(* Logix 5000 project; controller Test_PID 1769-L16ER-BB1B rev 32.13; software revision 32.02 *)

TASK MainTask (continuous, watchdog 500 ms) : MainProgram

MODULES
   Local : 1769-L16ER-BB1B (PointIO 0, rev 32.13)
      Analog_Input1 : 1734-IE4C (PointIO 3, rev 3.1, Input RPI 80 ms)
      Discrete_IO : Embedded (PointIO 1, rev 32.11, Output RPI 20 ms)
      Relay_Output1 : vendor 1 type 7 code 231 (PointIO 2, rev 3.1, Output RPI 20 ms)
END_MODULES

TYPE EM_ProtoRockySequence_Int :
STRUCT
   Tmr : TIMER[64];
   StepTmr : TIMER;   // Step Timer
   PrevStepNmbr : DINT;   // Previous Step Number
   Bool : BOOL[64];
   Step : BOOL[64];
   SeqCmplt : BOOL;
   SeqActv : BOOL;
   Adsorption_Mixing : BOOL;
   Adsorption_H2OAdsorption : BOOL;
   Purge : BOOL;
   Desorption_ReverseRegen : BOOL;
   Desorption_Deep_Regen : BOOL;
   Desorption_CO2HeatingTop : BOOL;
   Desorption_CO2HeatingBottom : BOOL;
   Desorption_CO2Vacuum : BOOL;
   Regeneration_N2Heatup : BOOL;
   Regeneration_N2Regeneration : BOOL;
   measure_Moisture : BOOL;
   Regeneration_Cooling : BOOL;
   CO2_Recirculation : BOOL;
   Steam : BOOL;
END_STRUCT
END_TYPE

TYPE EM_Sequence :
STRUCT
   StepNmbr : DINT;
   SecS : DINT;
   GallonS : REAL;   // Step Gallons
   GalTog : BOOL;   // Step Show Gallons Toggle
   FaultS : BOOL;   // Sequenc Fault Status
   RunS : BOOL;   // Sequence Active Status
END_STRUCT
END_TYPE

TYPE SeqSteps :
STRUCT
   Step1 : BOOL;
   Step2 : BOOL;
   Step3 : BOOL;
   Step4 : BOOL;
END_STRUCT
END_TYPE

TYPE SeqTimers :
STRUCT
   Timer1 : TIMER;
   Timer2 : TIMER;
   Timer3 : TIMER;
END_STRUCT
END_TYPE

TYPE SeqTransition :
STRUCT
   Condition1 : BOOL;
   Condition2 : BOOL;
   Condition3 : BOOL;
END_STRUCT
END_TYPE

ADD_ON_INSTRUCTION StateControl   (* revision 1.0 *)
VAR_INPUT
   AbortC : BOOL;   // Abort Command
   Alarm : BOOL;   // Alarm Status
   Complete : BOOL;   // Complete Status
   HoldC : BOOL;   // Hold Command
   OkToAbort : BOOL;   // OK to Abort
   OkToHold : BOOL;   // OK to Hold
   OkToRestart : BOOL;   // OK to Restart
   OkToStart : BOOL;   // OK to Start
   RestartC : BOOL;   // Restart Command
   StartC : BOOL;   // Start Command
END_VAR
VAR_OUTPUT
   ABORTING : BOOL; {access Read Only}   // Aborting
   AbortP : BOOL; {access Read Only}   // Abort Permissive
   HELD : BOOL; {access Read Only}   // Held
   HoldP : BOOL; {access Read Only}   // Hold Permissive
   IDLE : BOOL; {access Read Only}   // Idle
   RESTARTING : BOOL; {access Read Only}   // Restarting
   RestartP : BOOL; {access Read Only}   // Restart Permissive
   RUNNING : BOOL; {access Read Only}   // Running
   StartP : BOOL; {access Read Only}   // Start Permissive
END_VAR
VAR_INPUT
   WaitC : BOOL;   // Wait Command
END_VAR
VAR_OUTPUT
   WAITING : BOOL; {access Read Only}   // Waiting
   STARTED : BOOL; {access Read Only}   // Started
END_VAR
VAR
   AbortS : BOOL;   // Abort Status Oneshot
   RestartS : BOOL;   // Restart Status Oneshot
   HoldS : BOOL;   // Hold Status Oneshot
   StartS : BOOL;   // Start Status Oneshot
END_VAR

ROUTINE Logic   (* ladder *)
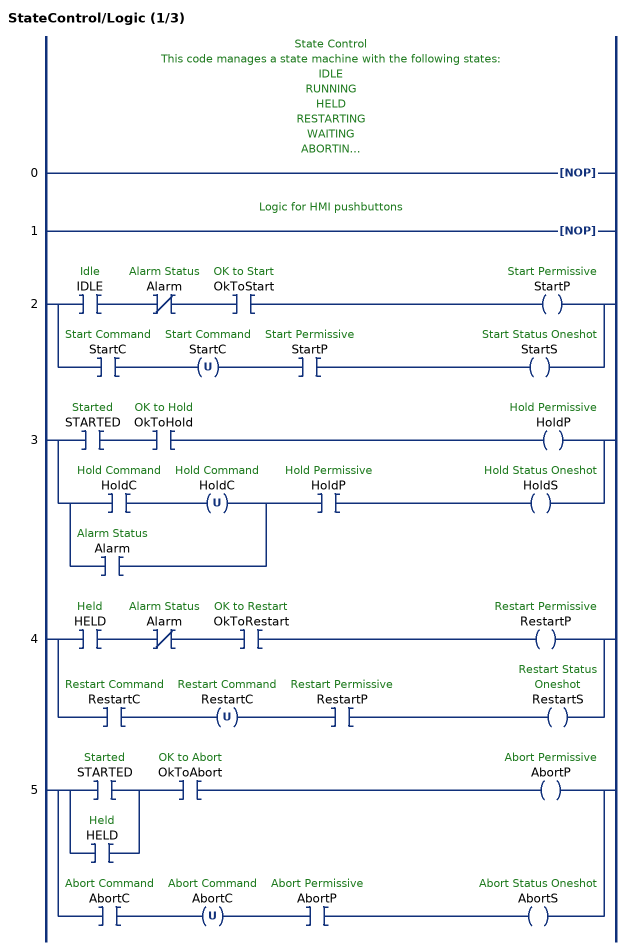
   // State Control
   // This code manages a state machine with the following states:
   // IDLE
   // RUNNING
   // HELD
   // RESTARTING
   // WAITING
   // ABORTING
   // The HMI interface consists of four pushbuttons:
   // Start
   // Hold
   // Restart
   // Abort
   // V1b - 7/15/11
   0: NOP();
   // Logic for HMI pushbuttons
   1: NOP();
   2: [XIC(IDLE) XIO(Alarm) XIC(OkToStart) OTE(StartP) ,XIC(StartC) OTU(StartC) XIC(StartP) OTE(StartS) ];
   3: [XIC(STARTED) XIC(OkToHold) OTE(HoldP) ,[XIC(HoldC) OTU(HoldC) ,XIC(Alarm) ] XIC(HoldP) OTE(HoldS) ];
   4: [XIC(HELD) XIO(Alarm) XIC(OkToRestart) OTE(RestartP) ,XIC(RestartC) OTU(RestartC) XIC(RestartP) OTE(RestartS) ];
   5: [[XIC(STARTED) ,XIC(HELD) ] XIC(OkToAbort) OTE(AbortP) ,XIC(AbortC) OTU(AbortC) XIC(AbortP) OTE(AbortS) ];
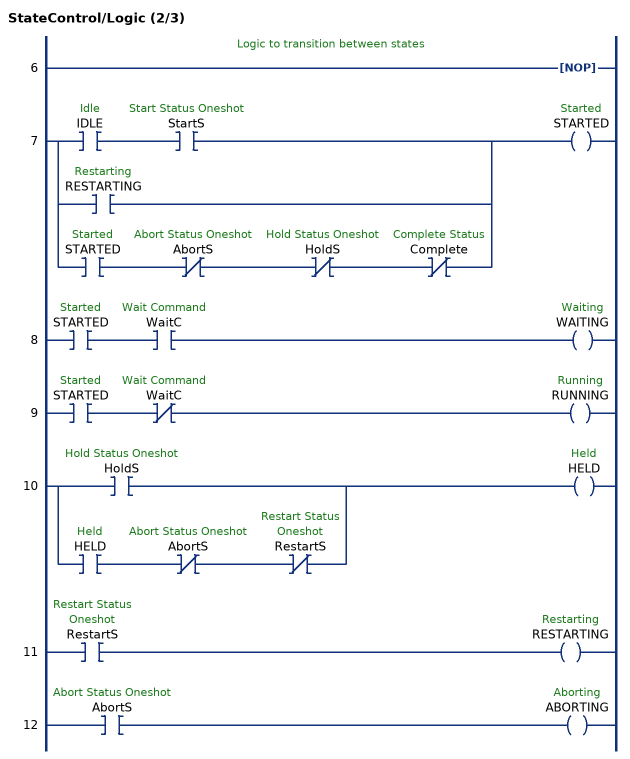
   // Logic to transition between states
   6: NOP();
   7: [[XIC(IDLE) XIC(StartS) ,XIC(RESTARTING) ] ,XIC(STARTED) XIO(AbortS) XIO(HoldS) XIO(Complete) ]OTE(STARTED);
   8: XIC(STARTED)XIC(WaitC)OTE(WAITING);
   9: XIC(STARTED)XIO(WaitC)OTE(RUNNING);
   10: [XIC(HoldS) ,XIC(HELD) XIO(AbortS) XIO(RestartS) ]OTE(HELD);
   11: XIC(RestartS)OTE(RESTARTING);
   12: XIC(AbortS)OTE(ABORTING);
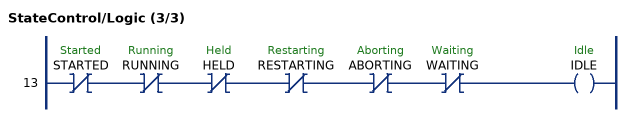
   13: XIO(STARTED)XIO(RUNNING)XIO(HELD)XIO(RESTARTING)XIO(ABORTING)XIO(WAITING)OTE(IDLE);
END_ROUTINE
END_ADD_ON_INSTRUCTION

VAR_GLOBAL   (* controller tags *)
   Alarm_Pumps_Flooding : BOOL;
   Alarm_Seq_Timeouts : BOOL;
   begin_Seq1_Start_PullDown_Tube : BOOL;
   begin_Seq3_Start_PullDown_Airlock : BOOL;
   begin_Seq4_Start_PumpDown_FS : BOOL;
   cmd_AbortPMS_HMI : BOOL;
   cmd_Close_AL_IsoV_Seq5 : BOOL;
   cmd_Close_Tube_IsoV_Seq5 : BOOL;
   cmd_FloodPumps_Seq5 : BOOL;
   cmd_Start_VentForeline : BOOL;
   cycle_type : BOOL;
   cycles_completed : DINT;
   cylcles_to_run : DINT := 3;
   emProtoRockyIISequence_i : EM_ProtoRockySequence_Int;
   emRockyIISequence : EM_Sequence;
   end_PumpsFlood_Seq : BOOL;
   fault_process : BOOL;
   Fault_Reset : BOOL;
   Fault_Seq_VentFL_Timeout : BOOL;
   hmi_abort_cycle : BOOL;
   hmi_auto_mode : BOOL := 1;
   hmi_cyles_to_run : DINT := 3;
   hmi_start_cycle : BOOL;
   hmi_stop_cycle : BOOL;
   interlockRun_VentForeline_Seq : BOOL := 1;
   interlockStart_VentForeline_Seq : BOOL := 1;
   man_seq1 : BOOL;
   man_seq11 : BOOL;
   man_seq12 : BOOL;
   man_seq13 : BOOL;
   man_seq2 : BOOL;
   man_seq3 : BOOL;
   mode_auto : BOOL := 1;
   ons_cycle_abort : BOOL;
   ons_cycle_completed : BOOL;
   ons_cycle_start : BOOL;
   ons_cycle_started : BOOL;
   ons_cycle_stop : BOOL;
   ons_seq3_done : BOOL;
   ONS_Seq_VentFL : BOOL[32];
   OpMode_isAuto : BOOL := 1;
   press_OLV_atVacuum : BOOL := 1;
   Pumps_areOFF : BOOL := 1;
   RockyIIState : StateControl := (OkToAbort := 1, OkToStart := 1, IDLE := 1, StartP := 1);
   seq11_done : BOOL;
   seq12_done : BOOL;
   seq13_done : BOOL;
   seq1_active : BOOL;
   seq1_done : BOOL;
   seq1_fault : INT;
   seq1_step : SeqSteps;
   seq1_tmr : SeqTimers := (Timer1.PRE := 10000, Timer2.PRE := 20000);
   seq1_trans : SeqTransition;
   seq2_active : BOOL;
   seq2_done : BOOL;
   seq2_fault : INT;
   seq2_step : SeqSteps;
   seq2_tmr : SeqTimers := (Timer1.PRE := 10000, Timer2.PRE := 20000);
   seq2_trans : SeqTransition;
   seq3_active : BOOL;
   seq3_done : BOOL;
   Seq_VentFL_Step : DINT;
   Seq_VentFL_StepNext : DINT;
   status_Airlock_IsoValve_isClosed : BOOL;
   status_IsoValve_isClosed : BOOL;
   status_Seq_FL_Vent_isRunning : BOOL;
   System_Faulted : BOOL;
   System_Safety_OK : BOOL := 1;
   tmr_seq_VentFL_Timeout : TIMER := (PRE := 10000);
   warning_process : BOOL;
END_VAR

PROGRAM MainProgram   (* main routine MainRoutine *)
VAR
   CO2_System_Delta_Des : DINT := 30;
   CO2Adsorption_CO2endThreshold : DINT := 10;
   PID_Loop_Call : BOOL;
   Test_Button : BOOL;
   Test_OnOff : BOOL;
   Timer_PID : TIMER := (PRE := 1000, ACC := 189, EN := 1, TT := 1);   // PID Timer
   tmr_OnOff : TIMER := (PRE := 60000);
   tmr_OnOff_Preset : DINT := 1;
END_VAR

ROUTINE Cycles_Test   (* ladder *)
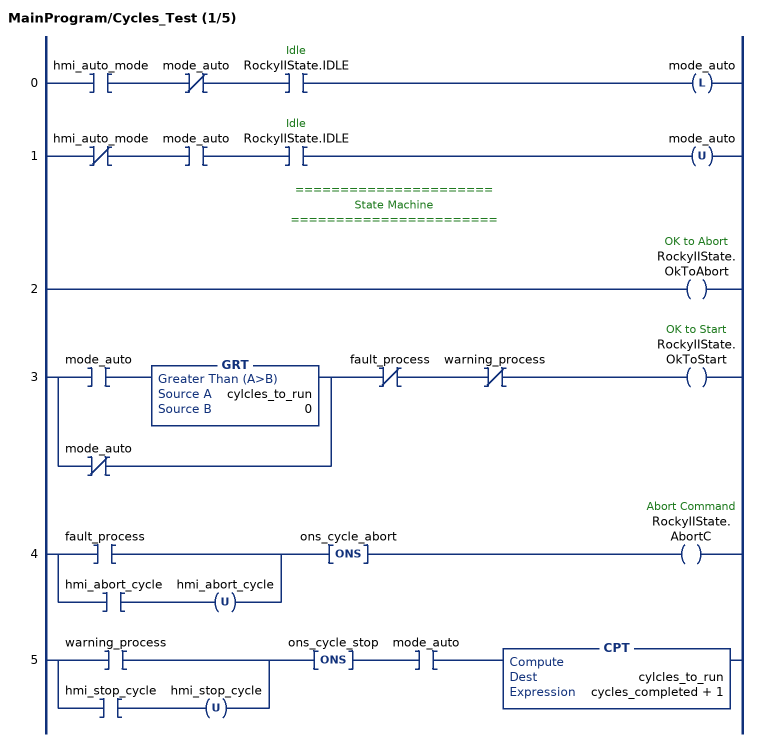
   0: XIC(hmi_auto_mode)XIO(mode_auto)XIC(RockyIIState.IDLE)OTL(mode_auto);
   1: XIO(hmi_auto_mode)XIC(mode_auto)XIC(RockyIIState.IDLE)OTU(mode_auto);
   // ======================
   // State Machine
   // =======================
   2: OTE(RockyIIState.OkToAbort);
   3: [XIC(mode_auto) GRT(cylcles_to_run,0) ,XIO(mode_auto) ]XIO(fault_process)XIO(warning_process)OTE(RockyIIState.OkToStart);
   4: [XIC(fault_process) ,XIC(hmi_abort_cycle) OTU(hmi_abort_cycle) ]ONS(ons_cycle_abort)OTE(RockyIIState.AbortC);
   5: [XIC(warning_process) ,XIC(hmi_stop_cycle) OTU(hmi_stop_cycle) ]ONS(ons_cycle_stop)XIC(mode_auto)CPT(cylcles_to_run,cycles_completed + 1);
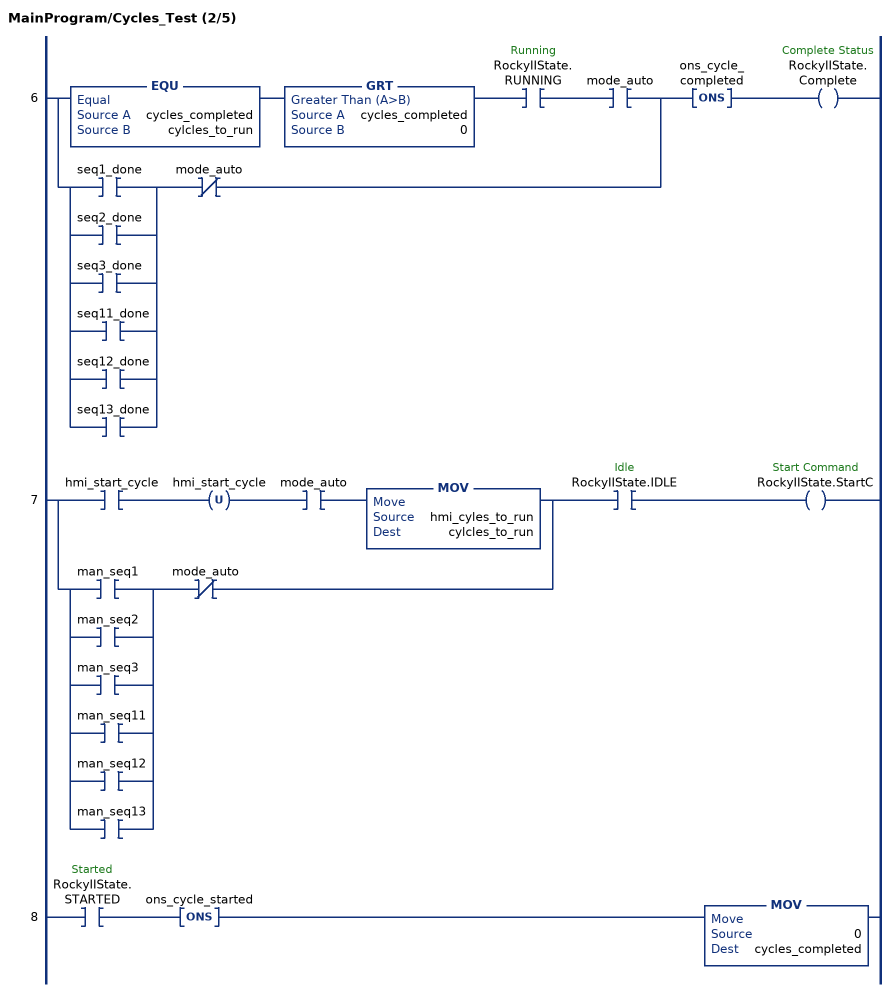
   6: [EQU(cycles_completed,cylcles_to_run) GRT(cycles_completed,0) XIC(RockyIIState.RUNNING) XIC(mode_auto) ,[XIC(seq1_done) ,XIC(seq2_done) ,XIC(seq3_done) ,XIC(seq11_done) ,XIC(seq12_done) ,XIC(seq13_done) ] XIO(mode_auto) ]ONS(ons_cycle_completed)OTE(RockyIIState.Complete);
   7: [XIC(hmi_start_cycle) OTU(hmi_start_cycle) XIC(mode_auto) MOV(hmi_cyles_to_run,cylcles_to_run) ,[XIC(man_seq1) ,XIC(man_seq2) ,XIC(man_seq3) ,XIC(man_seq11) ,XIC(man_seq12) ,XIC(man_seq13) ] XIO(mode_auto) ]XIC(RockyIIState.IDLE)OTE(RockyIIState.StartC);
   8: XIC(RockyIIState.STARTED)ONS(ons_cycle_started)MOV(0,cycles_completed);
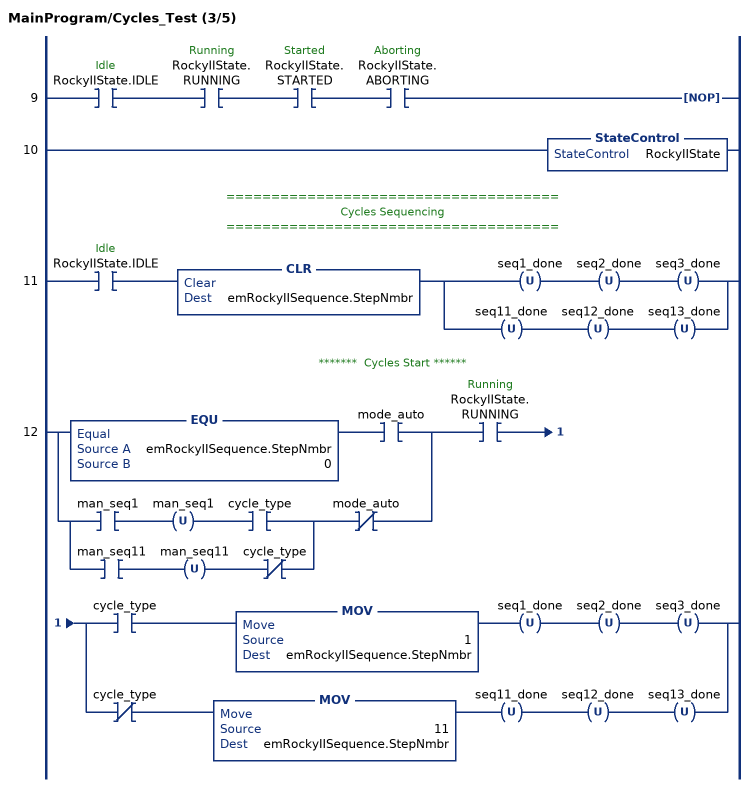
   9: XIC(RockyIIState.IDLE)XIC(RockyIIState.RUNNING)XIC(RockyIIState.STARTED)XIC(RockyIIState.ABORTING)NOP();
   10: StateControl(RockyIIState);
   // =====================================
   // Cycles Sequencing
   // =====================================
   11: XIC(RockyIIState.IDLE)CLR(emRockyIISequence.StepNmbr)[OTU(seq1_done) OTU(seq2_done) OTU(seq3_done) ,OTU(seq11_done) OTU(seq12_done) OTU(seq13_done) ];
   // *******  Cycles Start ******
   12: [EQU(emRockyIISequence.StepNmbr,0) XIC(mode_auto) ,[XIC(man_seq1) OTU(man_seq1) XIC(cycle_type) ,XIC(man_seq11) OTU(man_seq11) XIO(cycle_type) ] XIO(mode_auto) ]XIC(RockyIIState.RUNNING)[XIC(cycle_type) MOV(1,emRockyIISequence.StepNmbr) OTU(seq1_done) OTU(seq2_done) OTU(seq3_done) ,XIO(cycle_type) MOV(11,emRockyIISequence.StepNmbr) OTU(seq11_done) OTU(seq12_done) OTU(seq13_done) ];
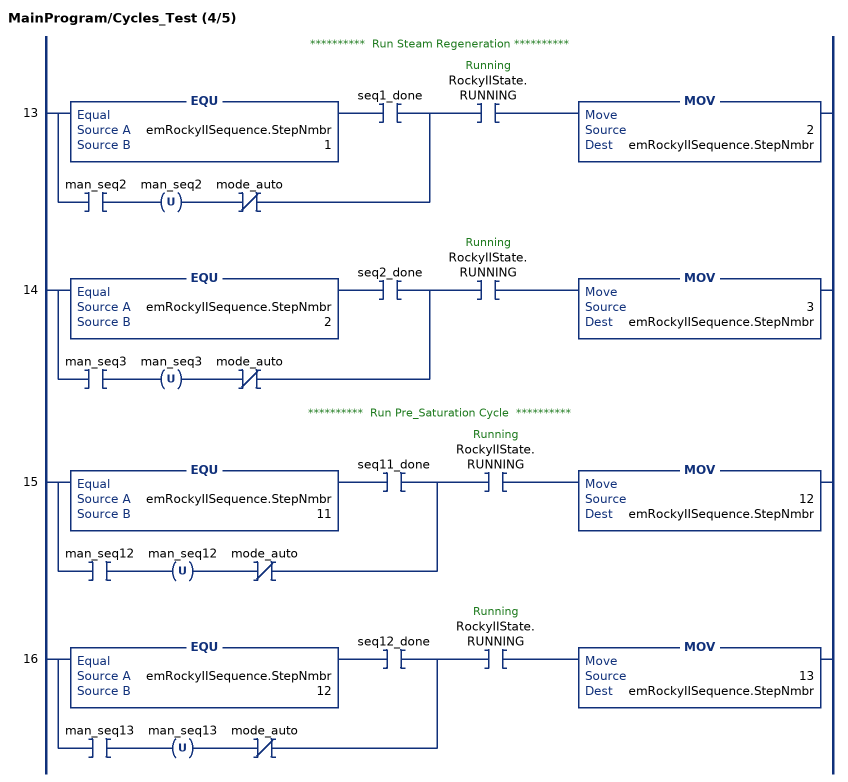
   // **********  Run Steam Regeneration **********
   13: [EQU(emRockyIISequence.StepNmbr,1) XIC(seq1_done) ,XIC(man_seq2) OTU(man_seq2) XIO(mode_auto) ]XIC(RockyIIState.RUNNING)MOV(2,emRockyIISequence.StepNmbr);
   14: [EQU(emRockyIISequence.StepNmbr,2) XIC(seq2_done) ,XIC(man_seq3) OTU(man_seq3) XIO(mode_auto) ]XIC(RockyIIState.RUNNING)MOV(3,emRockyIISequence.StepNmbr);
   // **********  Run Pre_Saturation Cycle  **********
   15: [EQU(emRockyIISequence.StepNmbr,11) XIC(seq11_done) ,XIC(man_seq12) OTU(man_seq12) XIO(mode_auto) ]XIC(RockyIIState.RUNNING)MOV(12,emRockyIISequence.StepNmbr);
   16: [EQU(emRockyIISequence.StepNmbr,12) XIC(seq12_done) ,XIC(man_seq13) OTU(man_seq13) XIO(mode_auto) ]XIC(RockyIIState.RUNNING)MOV(13,emRockyIISequence.StepNmbr);
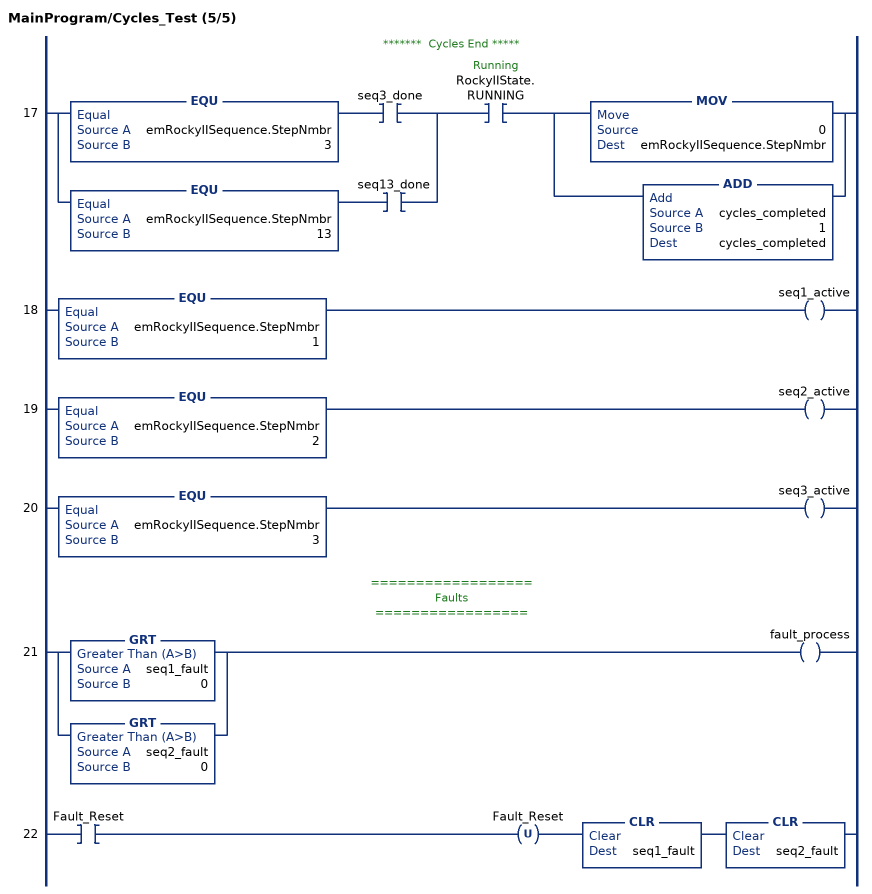
   // *******  Cycles End *****
   17: [EQU(emRockyIISequence.StepNmbr,3) XIC(seq3_done) ,EQU(emRockyIISequence.StepNmbr,13) XIC(seq13_done) ]XIC(RockyIIState.RUNNING)[MOV(0,emRockyIISequence.StepNmbr) ,ADD(cycles_completed,1,cycles_completed) ];
   18: EQU(emRockyIISequence.StepNmbr,1)OTE(seq1_active);
   19: EQU(emRockyIISequence.StepNmbr,2)OTE(seq2_active);
   20: EQU(emRockyIISequence.StepNmbr,3)OTE(seq3_active);
   // ==================
   // Faults
   // =================
   21: [GRT(seq1_fault,0) ,GRT(seq2_fault,0) ]OTE(fault_process);
   22: XIC(Fault_Reset)OTU(Fault_Reset)CLR(seq1_fault)CLR(seq2_fault);
END_ROUTINE

ROUTINE MainRoutine   (* ladder *)
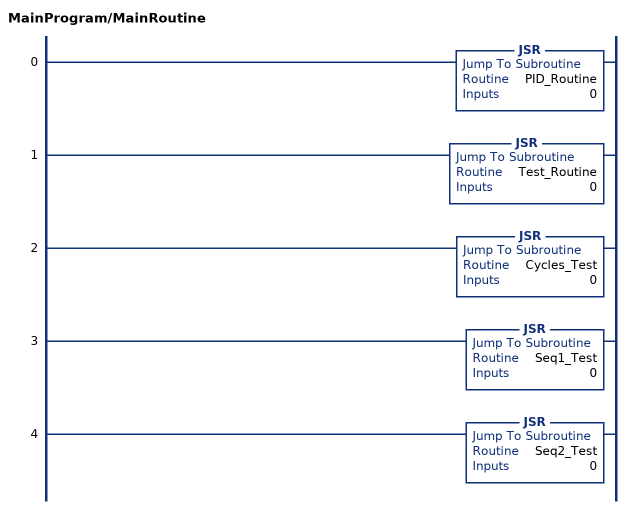
   0: JSR(PID_Routine,0);
   1: JSR(Test_Routine,0);
   2: JSR(Cycles_Test,0);
   3: JSR(Seq1_Test,0);
   4: JSR(Seq2_Test,0);
END_ROUTINE

ROUTINE PID_Routine   (* ladder *)
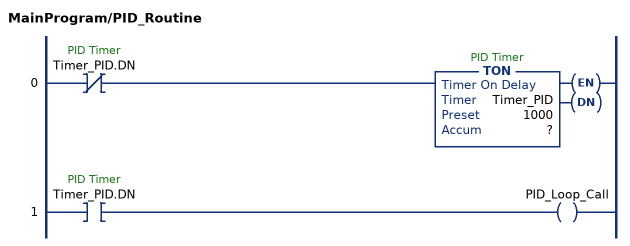
   0: XIO(Timer_PID.DN)TON(Timer_PID,?,?);
   1: XIC(Timer_PID.DN)OTE(PID_Loop_Call);
END_ROUTINE

ROUTINE Seq1_Test   (* ladder *)
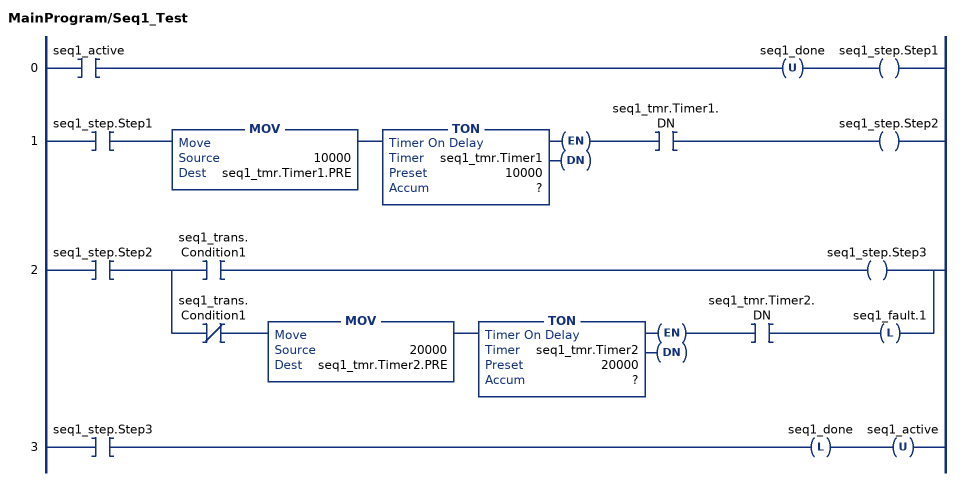
   0: XIC(seq1_active)OTU(seq1_done)OTE(seq1_step.Step1);
   1: XIC(seq1_step.Step1)MOV(10000,seq1_tmr.Timer1.PRE)TON(seq1_tmr.Timer1,?,?)XIC(seq1_tmr.Timer1.DN)OTE(seq1_step.Step2);
   2: XIC(seq1_step.Step2)[XIC(seq1_trans.Condition1) OTE(seq1_step.Step3) ,XIO(seq1_trans.Condition1) MOV(20000,seq1_tmr.Timer2.PRE) TON(seq1_tmr.Timer2,?,?) XIC(seq1_tmr.Timer2.DN) OTL(seq1_fault.1) ];
   3: XIC(seq1_step.Step3)OTL(seq1_done)OTU(seq1_active);
END_ROUTINE

ROUTINE Seq2_Test   (* ladder *)
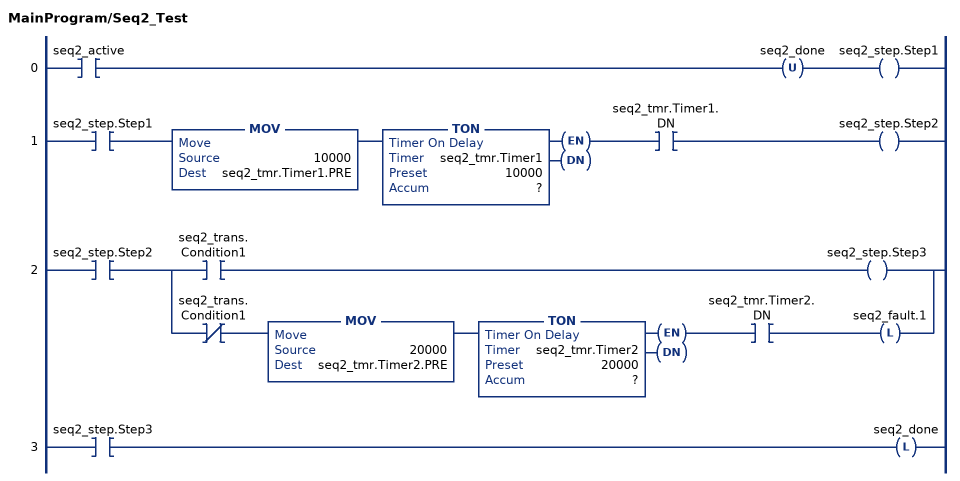
   0: XIC(seq2_active)OTU(seq2_done)OTE(seq2_step.Step1);
   1: XIC(seq2_step.Step1)MOV(10000,seq2_tmr.Timer1.PRE)TON(seq2_tmr.Timer1,?,?)XIC(seq2_tmr.Timer1.DN)OTE(seq2_step.Step2);
   2: XIC(seq2_step.Step2)[XIC(seq2_trans.Condition1) OTE(seq2_step.Step3) ,XIO(seq2_trans.Condition1) MOV(20000,seq2_tmr.Timer2.PRE) TON(seq2_tmr.Timer2,?,?) XIC(seq2_tmr.Timer2.DN) OTL(seq2_fault.1) ];
   3: XIC(seq2_step.Step3)OTL(seq2_done);
END_ROUTINE

ROUTINE Test_Routine   (* ladder *)
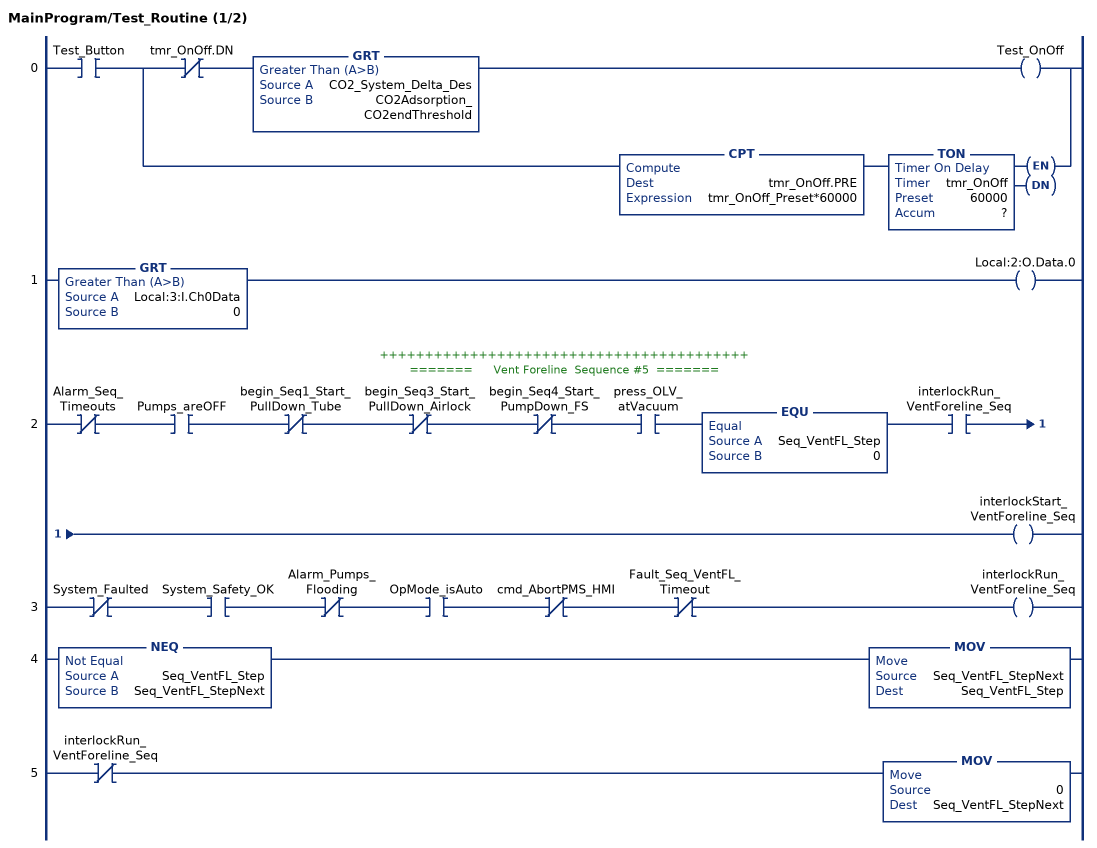
   0: XIC(Test_Button)[XIO(tmr_OnOff.DN) GRT(CO2_System_Delta_Des,CO2Adsorption_CO2endThreshold) OTE(Test_OnOff) ,CPT(tmr_OnOff.PRE,tmr_OnOff_Preset*60000) TON(tmr_OnOff,?,?) ];
   1: GRT(Local:3:I.Ch0Data,0)OTE(Local:2:O.Data.0);
   // +++++++++++++++++++++++++++++++++++++++++
   // =======      Vent Foreline  Sequence #5  =======
   2: XIO(Alarm_Seq_Timeouts)XIC(Pumps_areOFF)XIO(begin_Seq1_Start_PullDown_Tube)XIO(begin_Seq3_Start_PullDown_Airlock)XIO(begin_Seq4_Start_PumpDown_FS)XIC(press_OLV_atVacuum)EQU(Seq_VentFL_Step,0)XIC(interlockRun_VentForeline_Seq)OTE(interlockStart_VentForeline_Seq);
   3: XIO(System_Faulted)XIC(System_Safety_OK)XIO(Alarm_Pumps_Flooding)XIC(OpMode_isAuto)XIO(cmd_AbortPMS_HMI)XIO(Fault_Seq_VentFL_Timeout)OTE(interlockRun_VentForeline_Seq);
   4: NEQ(Seq_VentFL_Step,Seq_VentFL_StepNext)MOV(Seq_VentFL_StepNext,Seq_VentFL_Step);
   5: XIO(interlockRun_VentForeline_Seq)MOV(0,Seq_VentFL_StepNext);
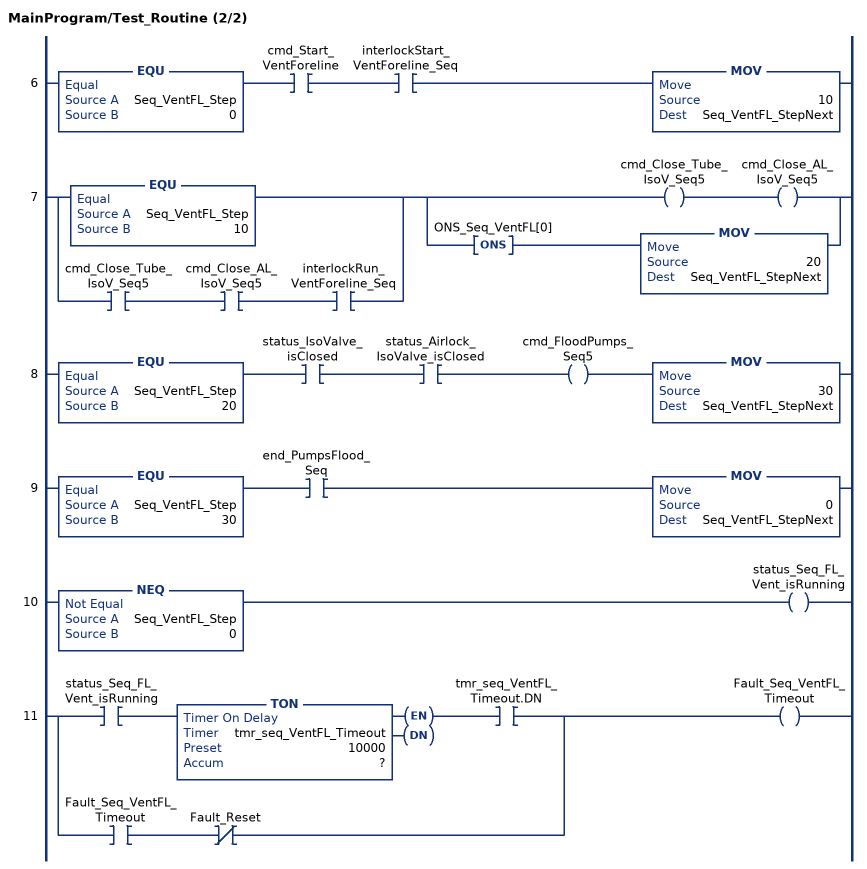
   6: EQU(Seq_VentFL_Step,0)XIC(cmd_Start_VentForeline)XIC(interlockStart_VentForeline_Seq)MOV(10,Seq_VentFL_StepNext);
   7: [EQU(Seq_VentFL_Step,10) ,XIC(cmd_Close_Tube_IsoV_Seq5) XIC(cmd_Close_AL_IsoV_Seq5) XIC(interlockRun_VentForeline_Seq) ][OTE(cmd_Close_Tube_IsoV_Seq5) OTE(cmd_Close_AL_IsoV_Seq5) ,ONS(ONS_Seq_VentFL[0]) MOV(20,Seq_VentFL_StepNext) ];
   8: EQU(Seq_VentFL_Step,20)XIC(status_IsoValve_isClosed)XIC(status_Airlock_IsoValve_isClosed)OTE(cmd_FloodPumps_Seq5)MOV(30,Seq_VentFL_StepNext);
   9: EQU(Seq_VentFL_Step,30)XIC(end_PumpsFlood_Seq)MOV(0,Seq_VentFL_StepNext);
   10: NEQ(Seq_VentFL_Step,0)OTE(status_Seq_FL_Vent_isRunning);
   11: [XIC(status_Seq_FL_Vent_isRunning) TON(tmr_seq_VentFL_Timeout,?,?) XIC(tmr_seq_VentFL_Timeout.DN) ,XIC(Fault_Seq_VentFL_Timeout) XIO(Fault_Reset) ]OTE(Fault_Seq_VentFL_Timeout);
END_ROUTINE
END_PROGRAM
